INTERFACE IPAProcessFunction EXTENDS IACComponent

PROPERTY ACState : ACStateEnum
GET
END_GET
SET
END_SET
END_PROPERTY

END_INTERFACE

(* stored: Version 1.1.0.1, ProductVersion 3.1.4024.6
   Itf IPAProcessFunction: Id {672626f8-954a-493c-924f-ece0de01c7e4}
   Property ACState: Id {cebbfa0e-c1f9-40d8-8238-0c74fe94c23f}
   Get Get: Id {c82ecdbb-fd0c-4ae5-b99c-cf3a6fde5bed}
   Set Set: Id {068047bc-9d25-4474-bed2-e090a934ad71} *)
